(*
SPDX-FileCopyrightText: © 2026 Oleksandr Tiutyk <trofimich@gmail.com>
SPDX-License-Identifier: MIT
License: https://opensource.org/license/mit
*)

(*!
<summary>Base for a file-content operation borrowing a manager-owned file resource.</summary>
<description>
Queue membership and resource binding do not transfer ownership. One owner drives the task. Keep the resource
owner alive while using its binding; an assigned reference alone does not prove acquisition. The manager
acquires the file before child execution and waits for child stopping before release. Removing a child from a
queue does not clear the binding. Reset from STOPPED clears it; READY Reset is a no-op. A removed READY child
must explicitly clear or replace its binding before the old owner is destroyed. Descendants overriding OnReset
must preserve binding cleanup. Descendants must finish native pending I/O during stopping before allowing the
parent to release the resource. Do not mutate borrowed resource data.
</description>
*)

FUNCTION_BLOCK ABSTRACT FileContentTask EXTENDS TOF_Tasks.Task IMPLEMENTS IFileContentTask
VAR
	_FileHandleResource : REFERENCE TO FileHandleResource;
END_VAR

(*!
<summary>File-content operations take the actual target from the bound resource</summary>
<description>
before submitting I/O, overriding any separately configured AmsNetId.
</description>
*)

{attribute 'monitoring' := 'call'}

PROPERTY ABSTRACT AmsNetId : Tc2_System.T_AmsNetID
GET
END_GET
SET
END_SET
END_PROPERTY

(*!
<summary>Reads the handle through the current borrowed resource binding.</summary>
<description>
Returns the default UINT when unbound. Does not establish acquisition; use only while the owning manager has
acquired the current file, and do not cache across release.
</description>
*)
{attribute 'monitoring' := 'call'}
PROPERTY FINAL FileHandle : UINT
GET
IF __ISVALIDREF(_FileHandleResource) THEN
	FileHandle := _FileHandleResource.FileHandle;
END_IF
END_GET
END_PROPERTY

(*!
<summary>Exposes the borrowed resource binding for this operation.</summary>
<description>
Returns an invalid reference when unbound. The owner must remain alive throughout access; an assigned
reference does not mean the file is acquired. Do not mutate borrowed data or close the handle independently.
</description>
*)
{attribute 'monitoring' := 'call'}
PROPERTY FINAL FileHandleResource : REFERENCE TO FileHandleResource
GET
IF __ISVALIDREF(_FileHandleResource) THEN
	FileHandleResource REF= _FileHandleResource;
END_IF
END_GET
END_PROPERTY

(*!
<summary>Copies the file path from the current resource binding.</summary>
<description>
Returns the default empty string when unbound. Reading requires the resource owner to remain alive; the path
is configuration and does not prove acquisition.
</description>
*)
{attribute 'monitoring' := 'call'}
PROPERTY FINAL FilePath : Tc2_System.T_MaxString
GET
IF __ISVALIDREF(_FileHandleResource) THEN
	FilePath := _FileHandleResource.FilePath;
END_IF
END_GET
END_PROPERTY

(*!
<summary>Clears the borrowed resource binding when a STOPPED child is reset.</summary>
<description>
Base Reset does not call this hook in READY. Overriding descendants must preserve this cleanup; it neither
closes the file nor removes the task from any queue.
</description>
*)
METHOD PROTECTED OnReset
_FileHandleResource REF= 0;
END_METHOD

(*!
<summary>Bind, replace or clear a borrowed resource only in READY; otherwise throw.</summary>
<description>
An invalid reference clears the binding. Reset a STOPPED task before rebinding. The caller must first remove
the task from any queue; READY alone does not mean it is unqueued. The resource owner must outlive its use by
this task. Queue removal does not clear this binding; READY Reset is a no-op. Clear or replace the binding
explicitly for a removed READY task before destroying the old resource owner.
</description>
*)

METHOD SetFileHandleResource
VAR_INPUT
	fileHandleResource : REFERENCE TO FileHandleResource;
END_VAR
IF NOT State.Ready THEN
	TOF_Core.Exceptions.ThrowStandard(
		sourceNamespaceName := NamespaceName,
		sourceClassName := ClassName,
		sourcePOUName := __POUNAME(),
		sourcePosition := __POSITION(),
		message := "FileHandleResource can only be assigned in READY state"
	);
END_IF

IF __ISVALIDREF(fileHandleResource) THEN
	_FileHandleResource REF= fileHandleResource;
ELSE
	_FileHandleResource REF= 0;
END_IF
END_METHOD

(*!
<summary>Configures the timeout passed to native operation requests.</summary>
<description>
Implementations apply this value to their native requests. Configure before execution and keep stable through
stopping; it is not a deadline for the entire task lifecycle.
</description>
*)
{attribute 'monitoring' := 'call'}
{attribute 'OPC.UA.DA.Property' := '1'}
{attribute 'OPC.UA.DA' := '1'}
PROPERTY ABSTRACT Timeout : TIME
GET
END_GET
SET
END_SET
END_PROPERTY

(*!
<summary>TRUE while the underlying file FB reports a pending request, including</summary>
<description>
cancellation wait. Reading has no side effects and does not indicate task lifecycle state or permission to
release the file resource.
</description>
*)

{attribute 'monitoring' := 'call'}

PROPERTY ABSTRACT FileOperationInProgress : BOOL
GET
END_GET
END_PROPERTY

END_FUNCTION_BLOCK

(* stored: Version 1.1.0.1
   POU FileContentTask: Id {e0edebf6-69ee-43f1-b0cd-ddf0e5a3f8d2}, SpecialFunc None
   Folder Members to override: Id {82ef782c-3b4a-42cb-882a-9ac933c30b73}
   Property AmsNetId: Id {ea169d19-fc59-4e8e-bfd6-f05e2562e2f5}
   Get Get: Id {75d6b396-2e53-497e-98ab-b2564567cddb}
   Set Set: Id {94e4e0c9-5dda-4170-b1e7-d631abb75196}
   Property FileHandle: Id {82868fbc-d80b-4342-95ff-b87334c6f19e}
   Get Get: Id {00add956-e3ac-47c9-87bd-7a30ec1b127b}
   Property FileHandleResource: Id {c52cc722-ac4c-47b4-8498-e198fd105426}
   Get Get: Id {52221dfa-f446-4fac-997a-fb4bbce2f4fa}
   Property FilePath: Id {5eefa187-b2a6-4167-b37b-7a1237013146}
   Get Get: Id {b73f03f2-fbb8-4ef6-a600-eed689f598d3}
   Method OnReset: Id {70ecd019-b2a8-415c-801a-36b22151de6e}
   Method SetFileHandleResource: Id {ae64e717-44da-42dc-b4c5-bc1e2b25543b}
   Property Timeout: Id {b3334de9-562b-4b05-996c-bb7c42bd5ba7}
   Get Get: Id {35a70dd8-7700-4e7d-a505-0a238f1252c8}
   Set Set: Id {833a7c4a-0925-4e43-965f-120e0cbe7c74}
   Property FileOperationInProgress: Id {041ef8d9-7239-4cbb-83d1-09970b80b63c}
   Get Get: Id {750d50bf-85e7-4858-8d7c-bf2631bde1be} *)
